// Elapsed seconds, measured in task scans.
//
// Carried over essentially unchanged - one of the few parts that
// needed nothing. Resolution is the task period, so a test shorter than one scan
// reports zero. That is honest: at this resolution there is nothing finer to say.
//
// Duration is reported, never asserted on. Scan counts are the reproducible
// measure across Windows, BSD, Linux RT and containers.
FUNCTION_BLOCK TestStopwatch
VAR
	_StartCycle		 : UDINT;
	_PreviousElapsed : LREAL;
	_IsRunning		 : BOOL;
END_VAR

(*
	No cyclic body. Elapsed is derived from the task's own cycle counter, so
	nothing has to be called every scan to keep it accurate.
*)

// Seconds since Start, or the frozen value once stopped.
PROPERTY Elapsed : LREAL
GET
VAR
	Cycles : UDINT;
END_VAR


IF NOT _IsRunning THEN
	Elapsed := _PreviousElapsed;
	RETURN;
END_IF

// Unsigned subtraction, so a wrapped cycle counter still yields the correct
// difference.
Cycles := TwinCAT_SystemInfoVarList._TaskInfo[GETCURTASKINDEXEX()].CycleCount - _StartCycle;

// CycleTime is in 100 ns units.
Elapsed := TO_LREAL(Cycles)
		 * TO_LREAL(TwinCAT_SystemInfoVarList._TaskInfo[GETCURTASKINDEXEX()].CycleTime)
		 / 10000000.0;
END_GET
END_PROPERTY

PROPERTY IsRunning : BOOL
GET
IsRunning := _IsRunning;
END_GET
END_PROPERTY

METHOD Reset
_PreviousElapsed := 0.0;
_StartCycle		 := 0;
_IsRunning		 := FALSE;
END_METHOD

// Restarts from zero. Starting an already-running stopwatch discards what it had.
METHOD Start
_PreviousElapsed := 0.0;
_StartCycle		 := TwinCAT_SystemInfoVarList._TaskInfo[GETCURTASKINDEXEX()].CycleCount;
_IsRunning		 := TRUE;
END_METHOD

// Freezes and returns the elapsed seconds. Stopping a stopped stopwatch returns
// what it already held rather than zero.
METHOD Stop : LREAL
IF _IsRunning THEN
	_PreviousElapsed := THIS^.Elapsed;
	_IsRunning		 := FALSE;
END_IF

Stop := _PreviousElapsed;
END_METHOD

END_FUNCTION_BLOCK

(* stored: Version 1.1.0.1, ProductVersion 3.1.4026.18
   POU TestStopwatch: Id {3cc4e536-9b8f-43c8-89e1-d34fc7913601}, SpecialFunc None
   Property Elapsed: Id {37f0ace4-1757-481a-ad3e-a4fa37d38ba3}
   Get Get: Id {35be167e-e1c6-435f-888b-28a2f00c94f8}
   Property IsRunning: Id {7f7506f8-e8f2-4e28-b0ce-125ead2977b6}
   Get Get: Id {15216e90-2da3-48b8-aeb7-9f8f243c274c}
   Method Reset: Id {35f80804-b9de-4097-8ee0-f7c2f5b74085}
   Method Start: Id {a29d664b-fea4-473d-a030-d5d168adf50e}
   Method Stop: Id {dd061033-f2d8-45d9-9594-7d8c30f50400} *)
